FUNCTION_BLOCK CYCLE_TIME (* Calculcates the Time passed since last Call. *)
  (* Standard: 61499-1; Description: Copyright (c) 2024 HR Agrartechnik GmbH This program and the accompanying materials are made available under the terms of the Eclipse Public License 2.0 which is available at https://www.eclipse.org/legal/epl-2.0/ SPDX-License-Identifier: EPL-2.0 *)
  (* Version 1.0, 2024-10-18, Franz Höpfinger, HR Agrartechnik GmbH *)
  PACKAGE utils::timing;
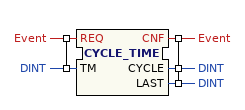
  EVENT_INPUT
    REQ WITH TM; (* Normal Execution Request *)
  END_EVENT
  EVENT_OUTPUT
    CNF WITH CYCLE, LAST; (* Execution Confirmation *)
  END_EVENT
  VAR_INPUT
    TM : DINT := 0; (* Current Call Time *)
  END_VAR
  VAR_OUTPUT
    CYCLE : DINT := 0; (* Cycle Time *)
    LAST : DINT := 0; (* Last Call Time *)
  END_VAR
  EC_STATES
    REQ : REQ -> CNF;
  END_STATES
  ALGORITHM REQ IN ST:
CYCLE := TM - LAST;
LAST := TM;
  END_ALGORITHM
END_FUNCTION_BLOCK
